FUNCTION_BLOCK GenIter
VAR
	_nIter		: UDINT;
	_bFirstLoop	: BOOL;
END_VAR

//FB_Init is always available implicitly and it is used primarily for initialization.
//The return value is not evaluated. For a specific influence, you can also declare the
//methods explicitly and provide additional code there with the standard initialization
//code. You can evaluate the return value.
METHOD FB_Init: BOOL
VAR_INPUT
    bInitRetains: BOOL; // TRUE: the retain variables are initialized (reset warm / reset cold)
    bInCopyCode: BOOL;  // TRUE: the instance will be copied to the copy code afterward (online change)

	nInit		: UDINT;  
END_VAR
_nIter := nInit;
END_METHOD

METHOD Get : UDINT
VAR_INPUT
END_VAR
Get := _nIter;
END_METHOD

METHOD Next : UDINT
VAR_INPUT
END_VAR
IF _bFirstLoop THEN
	_bFirstLoop := FALSE;
	Next := _nIter;
	RETURN;	
END_IF

_nIter := _nIter + 1;
Next := _nIter;
END_METHOD

METHOD Peek : UDINT
VAR_INPUT
END_VAR
Peek := _nIter + 1;
END_METHOD

METHOD PeekBack : UDINT
VAR_INPUT
END_VAR
PeekBack := _nIter - 1;
END_METHOD

METHOD Prev : UDINT
VAR_INPUT
END_VAR
IF _bFirstLoop THEN
	_bFirstLoop := FALSE;
	Next := _nIter;
	RETURN;	
END_IF

_nIter := _nIter - 1;
Next := _nIter;
END_METHOD

METHOD Set : UDINT
VAR_INPUT
	nNewValue	: UDINT;
END_VAR
_nIter := nNewValue;
Set := _nIter;
END_METHOD

END_FUNCTION_BLOCK

(* stored: Version 1.1.0.1
   POU GenIter: Id {bfb2d917-8d66-4d61-a6dd-fe69559f7b9a}, SpecialFunc None
   Method FB_init: Id {cccd5948-2a78-4a4d-b4df-a2a1d4bbf4e6}
   Method Get: Id {13848a90-780b-40f6-88a7-df0d2464868f}
   Method Next: Id {ae73b3bd-4943-4d15-837b-808bceca5e23}
   Method Peek: Id {89b11ba9-e7b9-43fb-9e1e-a9eee605994f}
   Method PeekBack: Id {46c79a93-25eb-44d7-94bc-583b1efe449f}
   Method Prev: Id {4f9115a7-ebbb-4986-abd8-b6e412678e6c}
   Method Set: Id {da18debc-0496-4d1f-a196-2ac754170463} *)
